FUNCTION_BLOCK FB_ErrorHandling
VAR_INPUT
	fbErrorBufferDistanceSensor : FB_ErrorBuffer;
	fbErrorBufferAccelerationSensor1 : FB_ErrorBuffer;
	fbErrorBufferAccelerationSensor2 : FB_ErrorBuffer;
END_VAR
VAR_OUTPUT
	bGoToSHUTDOWN : BOOL;
	bGoToERROR : BOOL;
END_VAR
VAR
	eState : eErrorHandlingSTM := eErrorhandlingSTM.CheckforErrorMessages;
	
	fbErrorBuffer : FB_MessageBuffer;
	fbWarningBuffer : FB_MessageBuffer;

	eErrorMessageDistanceSensor : eErrorList := eErrorList.NoError;	
	eErrorMessageAccelerationSensor1 : eErrorList := eErrorList.NoError;
	eErrorMessageAccelerationSensor2 : eErrorList := eErrorList.NoError;
	
	sMessage : STRING;
	bCriticalError : BOOL;
	i : UDINT;
END_VAR

//ErrorHandlingSTM
CASE eState OF
	eErrorhandlingSTM.CheckforErrorMessages:
		bGoToSHUTDOWN := FALSE;
		bGoToERROR := FALSE;
		IF MainControl.fbServiceModule.eCondition = eConditionCheck.READY AND MainControl.fbLevitationSystem.eCondition = eConditionCheck.READY AND MainControl.fbGuidanceSystem.eCondition = eConditionCheck.READY THEN
			eState := eErrorhandlingSTM.CheckforErrorMessages;
		ELSE
			//DistanceSensor
			IF fbErrorBufferDistanceSensor.getNumberOfMessages > 0 THEN
				fbErrorBufferDistanceSensor.GetAndRemoveErrorMessage(eErrorMessage => eErrorMessageDistanceSensor);
				CASE eErrorMessageDistanceSensor OF
					eErrorList.CommunicationError:
						sMessage := TO_STRING(eWarningMessages.DistanceSensor_CommunicationError);
						fbWarningBuffer.AddMessage(eMessage := sMessage);
					eErrorList.OutOfRange:
						sMessage := TO_STRING(eWarningMessages.DistanceSensor_OutOfRange);
						fbWarningBuffer.AddMessage(eMessage := sMessage);
				END_CASE
			END_IF
			//AccelerationSensor1
			IF fbErrorBufferAccelerationSensor1.getNumberOfMessages > 0 THEN
				fbErrorBufferAccelerationSensor1.GetAndRemoveErrorMessage(eErrorMessage => eErrorMessageAccelerationSensor1);
				CASE eErrorMessageAccelerationSensor1 OF
					eErrorList.OutOfRange:
						sMessage := TO_STRING(eWarningMessages.IMU1_OutOfRange);
						fbWarningBuffer.AddMessage(eMessage := sMessage);
					eErrorList.CommunicationError:
						sMessage := TO_STRING(eErrorMessages.IMU1_CommunicationError);
						fbErrorBuffer.AddMessage(eMessage := sMessage);	
						bCriticalError := TRUE;	
				END_CASE
			END_IF
			//AccelerationSensor2
			IF fbErrorBufferAccelerationSensor2.getNumberOfMessages > 0 THEN
				fbErrorBufferAccelerationSensor2.GetAndRemoveErrorMessage(eErrorMessage => eErrorMessageAccelerationSensor2);
				CASE eErrorMessageAccelerationSensor2 OF
					eErrorList.OutOfRange:
						sMessage := TO_STRING(eWarningMessages.IMU2_OutOfRange);
						fbWarningBuffer.AddMessage(eMessage := sMessage);
					eErrorList.CommunicationError:
						sMessage := TO_STRING(eErrorMessages.IMU2_CommunicationError);
						fbErrorBuffer.AddMessage(eMessage := sMessage);	
						bCriticalError := TRUE;	
				END_CASE
			END_IF
			
			IF bCriticalError THEN
				eState := eErrorHandlingSTM.ShowError;
				bCriticalError := FALSE;
			ELSE
				eState := eErrorHandlingSTM.ShowWarning;
			END_IF
		
		END_IF
		
	eErrorhandlingSTM.ShowWarning:
		FOR i:=0 TO fbWarningBuffer.getNumberOfMessages-1 BY 1 DO
			fbWarningBuffer.GetAndRemoveMessage(eMessage => MyGVLData.sWarningMessage[i]);
		END_FOR
		eState := eErrorHandlingSTM.CheckforErrorMessages;
		
	eErrorhandlingSTM.ShowError:
		FOR i:=0 TO fbErrorBuffer.getNumberOfMessages-1 BY 1 DO
			fbErrorBuffer.GetAndRemoveMessage(eMessage => MyGVLData.sErrorMessage[i]);
		END_FOR
		
		IF MainControl.eMainState = eMainStateMachine.OPERATIONAL THEN
			bGoToSHUTDOWN := TRUE;
		ELSIF MainControl.eMainState = eMainStateMachine.READY THEN
			bGoToERROR := TRUE;
		END_IF
		eState := eErrorHandlingSTM.CheckforErrorMessages;
END_CASE

END_FUNCTION_BLOCK

(* stored: Version 1.1.0.1, ProductVersion 3.1.4024.12
   POU FB_ErrorHandling: Id {e04ced6c-c731-48e4-8d82-f7134c556dd6}, SpecialFunc None *)
